FUNCTION_BLOCK BUGWORK (* Tests parsing and generation of base-16 numbers *)
  (* Standard: 61499-1 *)
  (* Version 0.1, 2004-05-02, JHC, Rockwell Automation, Moved to fb.rt.test. *)
  (* Version 0.0, 2002-10-27, JHC, Rockwell Automation *)
  (* Compiler header: package fb.rt.test; *)
  (* Compiler Java Sun JDK 1.3.1 *)
  (* Compiler Java IBM Jikes 1.06 *)
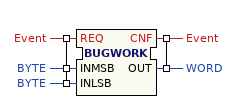
  EVENT_INPUT
    REQ WITH INMSB, INLSB;
  END_EVENT
  EVENT_OUTPUT
    CNF WITH OUT;
  END_EVENT
  VAR_INPUT
    INMSB : BYTE;
    INLSB : BYTE;
  END_VAR
  VAR_OUTPUT
    OUT : WORD;
  END_VAR
  VAR
    MASK : WORD := 16#00FF;
  END_VAR
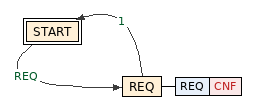
  EC_STATES
    START; (* Initial State *)
    REQ : REQ -> CNF; (* Normal execution *)
  END_STATES
  EC_TRANSITIONS
    START TO REQ := REQ;
    REQ TO START := 1;
  END_TRANSITIONS
  ALGORITHM REQ IN ST:
OUT:=INMSB*256+(INLSB&MASK);
  END_ALGORITHM
END_FUNCTION_BLOCK
